// SIMATIC S7-200 project (STEP 7-Micro/WIN), CPU 224XP REL 02.00

ORGANIZATION_BLOCK ?÷:OB1
TITLE=程序注解
BEGIN
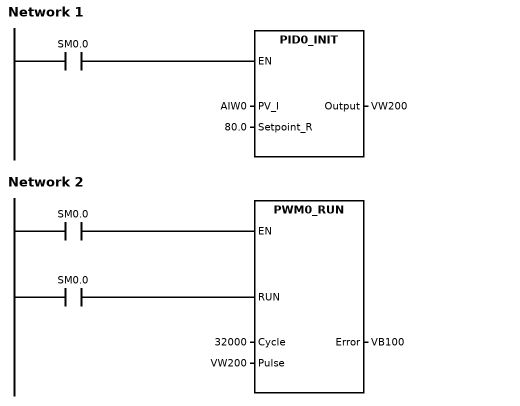
Network 1
LD     SM0.0
CALL   PID0_INIT:SBR1, AIW0, 80.0, VW200
Network 2
// (network saved uncompiled; LAD cells follow)
// row 0: c0 -| |- SM0.0  c1 --  c2 [PWM0_RUN EN:=power@row0, RUN:=power@row1, Cycle:=32000, Pulse:=VW200, Error=>VB100]
// row 1: c0 -| |- SM0.0  c1 --  c2 [box]
// row 2: c2 [box]
END_ORGANIZATION_BLOCK

// SBR1: protected block, not included

// SBR2: protected block, not included

// INT1: protected block, not included

// (further data pages could not be read)
